FUNCTION_BLOCK SchieberControl_AX (* Basic FB with Schieber ECC (AX Adapter Version) *)
  (* Standard: 61499-2; Description: Copyright (c) 2025 HR Agrartechnik GmbH This program and the accompanying materials are made available under the terms of the Eclipse Public License 2.0 which is available at https://www.eclipse.org/legal/epl-2.0/ SPDX-License-Identifier: EPL-2.0 *)
  (* Version 1.0, 2025-06-03, Franz Höpfinger, HR Agrartechnik GmbH *)
  PACKAGE logiBUS::utils::sequence::schieber;
  IMPORT logiBUS::utils::sequence::schieber::const::START;
  IMPORT logiBUS::utils::sequence::schieber::const::STATES;
  IMPORT logiBUS::utils::sequence::schieber::const::iSTATES;
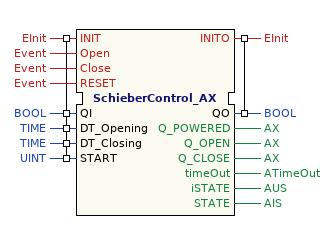
  EVENT_INPUT
    INIT : EInit WITH QI, DT_Opening, DT_Closing, START; (* Set all Values. Initialization Request. De-Init is not  fully supported. *)
    Open; (* Open *)
    Close; (* Close *)
    RESET; (* Reset to unknown State *)
  END_EVENT
  EVENT_OUTPUT
    INITO : EInit WITH QO; (* All Values have been Set. Initialization Confirm. *)
  END_EVENT
  VAR_INPUT
    QI : BOOL; (* Input event qualifier *)
    DT_Opening : TIME; (* TIME Setting *)
    DT_Closing : TIME; (* TIME Setting *)
    START : UINT := START::STARTUnknown;
  END_VAR
  VAR_OUTPUT
    QO : BOOL; (* Output event qualifier *)
  END_VAR
  PLUGS
    Q_POWERED : adapter::types::unidirectional::AX; (* Actuate "Open" Valve for Pneumatic *)
    Q_OPEN : adapter::types::unidirectional::AX; (* Actuate "Open" Valve *)
    Q_CLOSE : adapter::types::unidirectional::AX; (* Actuate "Close" Valve *)
    timeOut : iec61499::events::ATimeOut; (* timeOut Adapter *)
    iSTATE : adapter::types::unidirectional::AUS;
    STATE : adapter::types::unidirectional::AIS;
  END_PLUGS
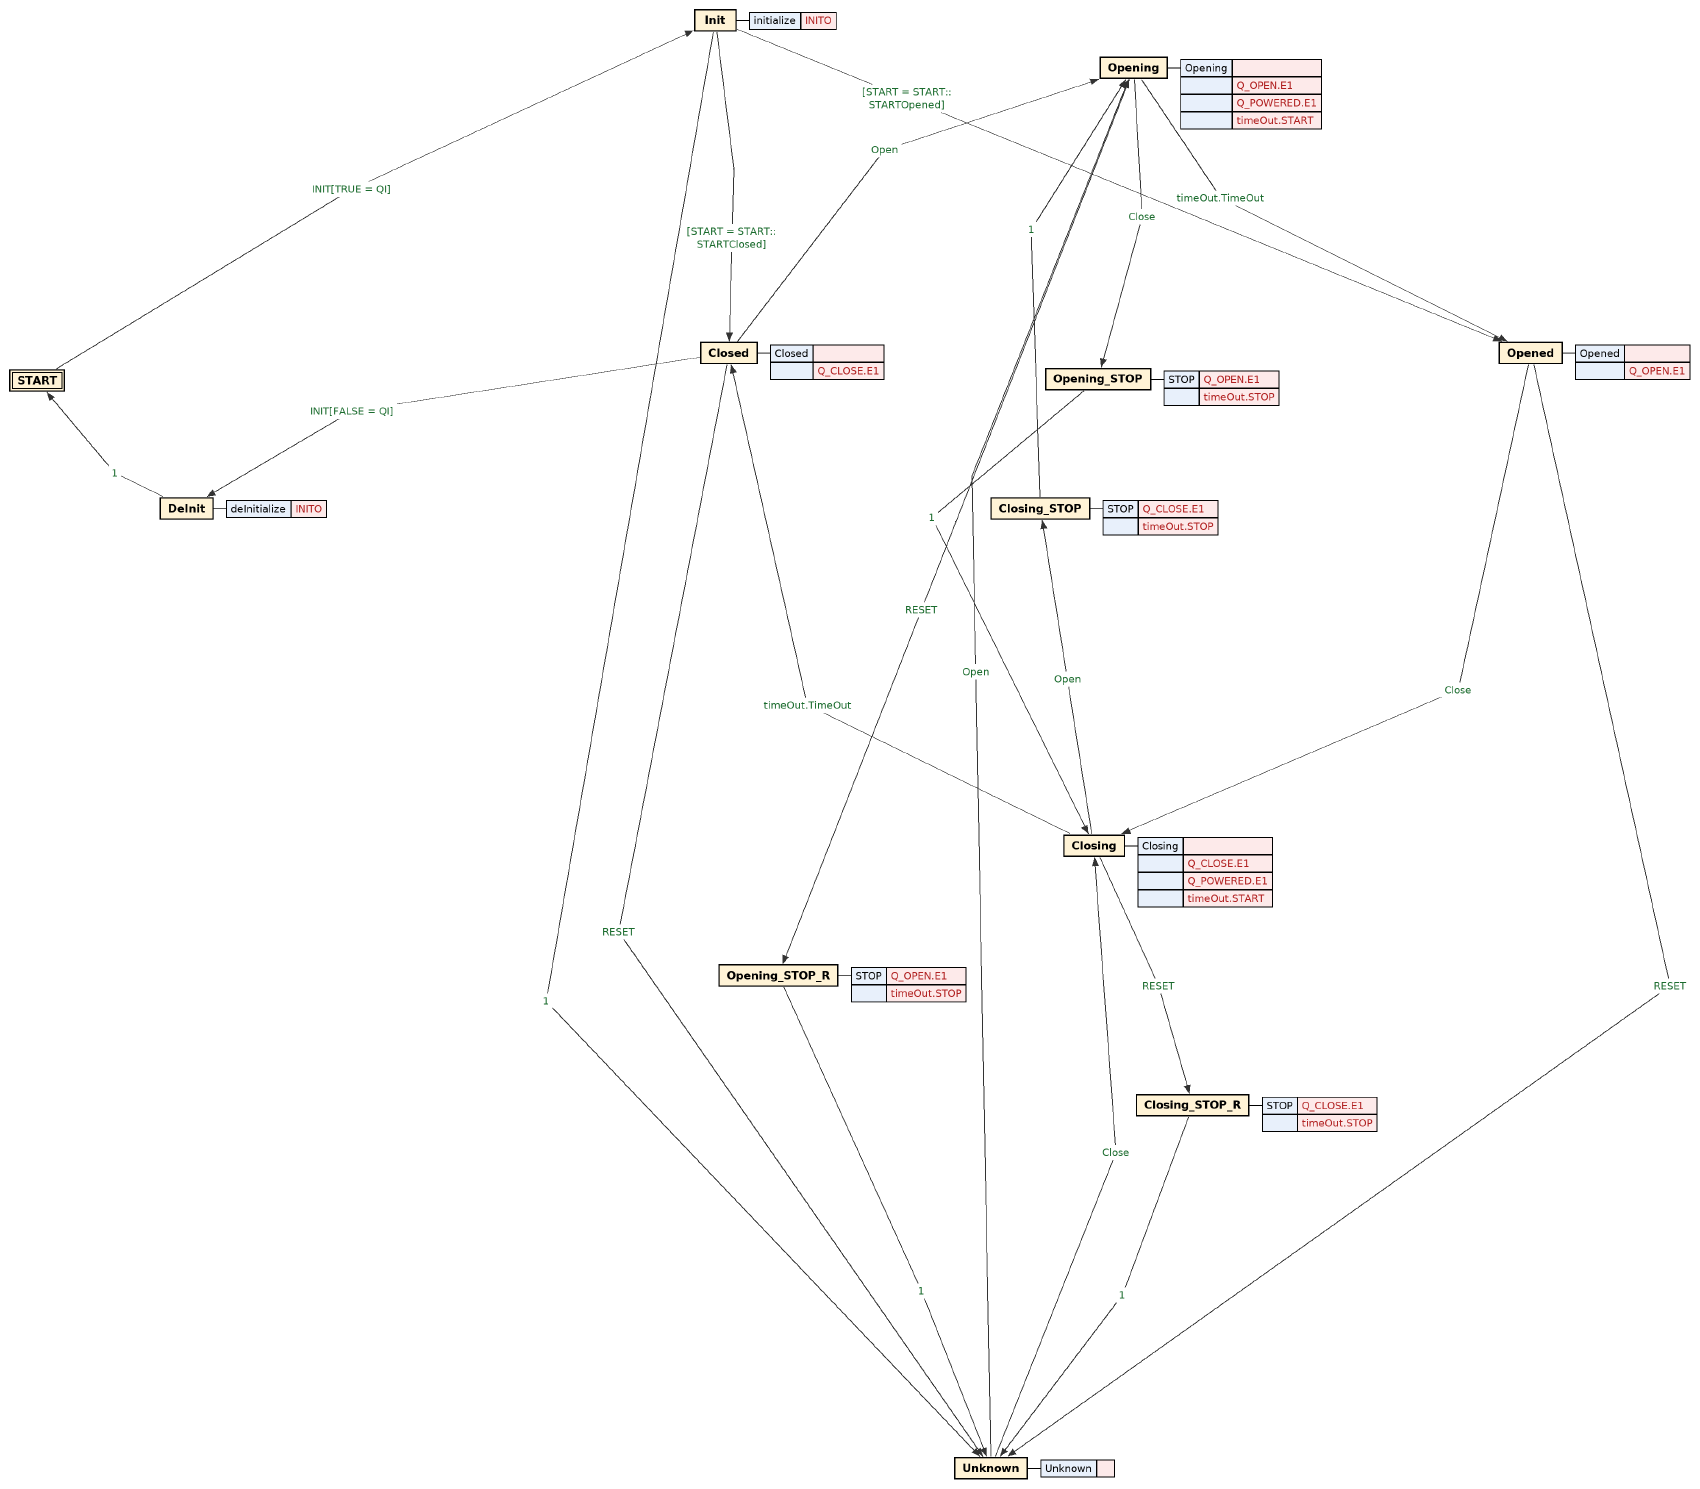
  EC_STATES
    START; (* Initial State *)
    Closed : Closed, -> Q_CLOSE.E1;
    DeInit : deInitialize -> INITO;
    Opened : Opened, -> Q_OPEN.E1;
    Closing : Closing, -> Q_CLOSE.E1, -> Q_POWERED.E1, -> timeOut.START;
    Opening : Opening, -> Q_OPEN.E1, -> Q_POWERED.E1, -> timeOut.START;
    Opening_STOP : STOP -> Q_OPEN.E1, -> timeOut.STOP;
    Closing_STOP : STOP -> Q_CLOSE.E1, -> timeOut.STOP;
    Unknown : Unknown;
    Opening_STOP_R : STOP -> Q_OPEN.E1, -> timeOut.STOP;
    Closing_STOP_R : STOP -> Q_CLOSE.E1, -> timeOut.STOP;
    Init : initialize -> INITO;
  END_STATES
  EC_TRANSITIONS
    DeInit TO START := 1;
    Closed TO Opening := Open;
    Closed TO DeInit := INIT[FALSE = QI];
    Opening TO Opened := timeOut.TimeOut;
    Opened TO Closing := Close;
    Closing TO Closed := timeOut.TimeOut;
    Opening TO Opening_STOP := Close;
    Closing TO Closing_STOP := Open;
    Opening_STOP TO Closing := 1;
    Closing_STOP TO Opening := 1;
    Opened TO Unknown := RESET;
    Closed TO Unknown := RESET;
    Opening TO Opening_STOP_R := RESET;
    Closing TO Closing_STOP_R := RESET;
    Opening_STOP_R TO Unknown := 1;
    Closing_STOP_R TO Unknown := 1;
    Unknown TO Opening := Open;
    Unknown TO Closing := Close;
    Init TO Closed := [START = START::STARTClosed];
    Init TO Opened := [START = START::STARTOpened];
    Init TO Unknown := 1;
    START TO Init := INIT[TRUE = QI];
  END_TRANSITIONS
  ALGORITHM initialize IN ST:
QO := QI;
  END_ALGORITHM
  ALGORITHM deInitialize IN ST:
QO := BOOL#FALSE;
  END_ALGORITHM
  ALGORITHM Closed IN ST:
STATE.D1 := STATES::Closed;
iSTATE.D1 := iSTATES::Closed;
Q_POWERED.D1 := BOOL#FALSE;
Q_OPEN.D1 := BOOL#FALSE;
Q_CLOSE.D1 := BOOL#FALSE;
  END_ALGORITHM
  ALGORITHM Opening IN ST:
STATE.D1 := STATES::Opening;
iSTATE.D1 := iSTATES::Opening;
timeOut.DT := DT_Opening;
Q_POWERED.D1 := BOOL#TRUE;
Q_OPEN.D1 := BOOL#TRUE;
Q_CLOSE.D1 := BOOL#FALSE;
  END_ALGORITHM
  ALGORITHM Opened IN ST:
STATE.D1 := STATES::Opened;
iSTATE.D1 := iSTATES::Opened;
Q_POWERED.D1 := BOOL#TRUE;
Q_OPEN.D1 := BOOL#FALSE;
Q_CLOSE.D1 := BOOL#FALSE;
  END_ALGORITHM
  ALGORITHM Closing IN ST:
STATE.D1 := STATES::Closing;
iSTATE.D1 := iSTATES::Closing;
timeOut.DT := DT_Closing;
Q_POWERED.D1 := BOOL#FALSE;
Q_OPEN.D1 := BOOL#FALSE;
Q_CLOSE.D1 := BOOL#TRUE;
  END_ALGORITHM
  ALGORITHM STOP IN ST:
// Powered_unchanged
Q_OPEN.D1 := BOOL#FALSE;
Q_CLOSE.D1 := BOOL#FALSE;
  END_ALGORITHM
  ALGORITHM Unknown IN ST:
STATE.D1 := STATES::Unknown;
iSTATE.D1 := iSTATES::Unknown;
Q_POWERED.D1 := BOOL#FALSE;
Q_OPEN.D1 := BOOL#FALSE;
Q_CLOSE.D1 := BOOL#FALSE;
  END_ALGORITHM
END_FUNCTION_BLOCK
